INTERFACE I_HaveParameters EXTENDS __SYSTEM.IQueryInterface

METHOD AddDataAsParameter
VAR_INPUT
	Name : T_MAXSTRING;
	Data : I_Datatype;
END_VAR
END_METHOD

METHOD AddParameter
VAR_INPUT
	Parameter : I_Parameter;
END_VAR
END_METHOD

METHOD PUBLIC GetParameters : I_Parameters
VAR_INPUT
END_VAR
END_METHOD

METHOD PUBLIC TryGetParameterByName : BOOL
VAR_INPUT
	Name : T_MAXSTRING;
	Destination : REFERENCE TO I_Parameter;
END_VAR
END_METHOD

END_INTERFACE

(* stored: Version 1.1.0.1, ProductVersion 3.1.4024.12
   Itf I_HaveParameters: Id {c5806033-3adc-0f99-304c-e569fa5b2b9f}
   Method AddDataAsParameter: Id {f6ff44a2-87ca-47cc-a380-2e4d25944377}
   Method AddParameter: Id {629b0de3-c6af-0abc-2e2a-6709cf7d0165}
   Method GetParameters: Id {83aea430-01cb-0969-3ea6-7616f2695ec6}
   Method TryGetParameterByName: Id {54f7a4bd-70df-0013-2d50-559760c48b28} *)
